// Mitsubishi GX Works2 project: 241021_자동화설비기능사_과제1   PLC: Q03UDV

PROGRAM TEST
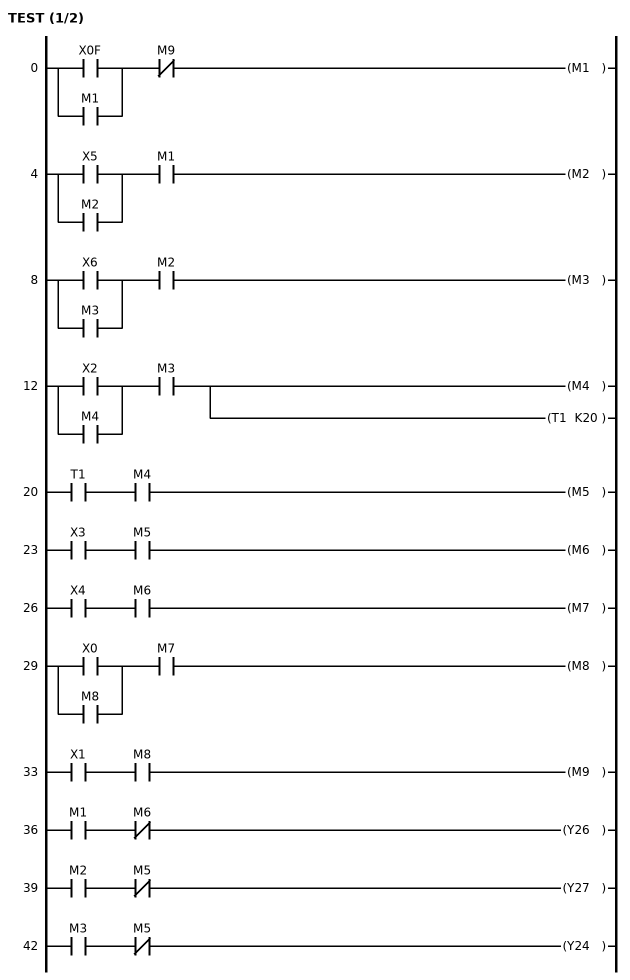
0     LD      X0F
      OR      M1
      ANI     M9
      OUT     M1
4     LD      X5
      OR      M2
      AND     M1
      OUT     M2
8     LD      X6
      OR      M3
      AND     M2
      OUT     M3
12    LD      X2
      OR      M4
      AND     M3
      OUT     M4
      OUT     T1 K20
20    LD      T1
      AND     M4
      OUT     M5
23    LD      X3
      AND     M5
      OUT     M6
26    LD      X4
      AND     M6
      OUT     M7
29    LD      X0
      OR      M8
      AND     M7
      OUT     M8
33    LD      X1
      AND     M8
      OUT     M9
36    LD      M1
      ANI     M6
      OUT     Y26
39    LD      M2
      ANI     M5
      OUT     Y27
42    LD      M3
      ANI     M5
      OUT     Y24
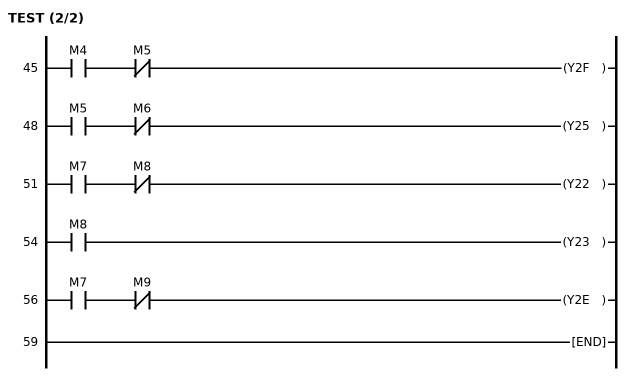
45    LD      M4
      ANI     M5
      OUT     Y2F
48    LD      M5
      ANI     M6
      OUT     Y25
51    LD      M7
      ANI     M8
      OUT     Y22
54    LD      M8
      OUT     Y23
56    LD      M7
      ANI     M9
      OUT     Y2E
59    END
END_PROGRAM
